FUNCTION_BLOCK SkidMagazine EXTENDS MaterialHolder
VAR_OUTPUT
	occupied : ARRAY[1..GVL.maxQueue] OF BOOL;
	
	inPosition1 AT %I* : BOOL;
	inPosition2 AT %I* : BOOL;
END_VAR

METHOD setOccupancy : BOOL
VAR_INPUT
	i : INT;
	occupancy : BOOL;
END_VAR
occupied[i] := occupancy;
END_METHOD

END_FUNCTION_BLOCK

(* stored: Version 1.1.0.1, ProductVersion 3.1.4024.11
   POU SkidMagazine: Id {3fc5a5bc-3ce1-4dc4-bdfd-362d2487d9e5}, SpecialFunc None
   Method setOccupancy: Id {2d1b747f-ab4a-4753-9254-fde4bc0bb760} *)
